// TIA Portal V17 export
// export: Created 2023-12-22T15:05:34.6100322Z, ExportSetting WithDefaults, DisplayName Totally Integrated Automation Portal, DisplayVersion V17, DisplayName TIA Portal Openness, DisplayVersion V17, DisplayName TIA Portal Version Control Interface, DisplayVersion V17, DisplayName STEP 7 Professional, DisplayVersion V17, DisplayName STEP 7 Safety, DisplayVersion V17, DisplayName WinCC Advanced, DisplayVersion V17
DATA_BLOCK "DB_Comm"   // DB99
{ S7_Optimized_Access := 'FALSE' }
VERSION : 0.1
// stored: AutoNumber false, DBAccessibleFromOPCUA true, IsOnlyStoredInLoadMemory false, IsWriteProtectedInAS false
   VAR RETAIN
      Input : Struct
         Line : Array[0..7] of Struct   // Линии
            Start : Bool;   // Дистанционный старт линии
            Mode : Bool;   // 0 - без разбавления, 1 - с разбавлением
            D : Real;   // Доза линии
         END_STRUCT;
         Pump : Array[1..10] of Struct   // Насосы
            Reserv : Bool;   // 0 - насос основной, 1 - насос резервный
            Line_Main : Int;   // Главная линия насоса
            Line_Reserve : Int;   // Резервная линия насоса
         END_STRUCT;
         Input_PolyMix_1 : "PolyMix_Input";
         Input_PolyMix_2 : "PolyMix_Input";
         Flow_LSAU_1 : Real := 1314.753;   // м3/ч
         Flow_LSAU_2 : Real := 0.0;
         Reset_All : Bool := FALSE;
         PolyMix_1_Source_BK1 : Bool := FALSE;   // Жидкий полимикс - качает с бака 1
         PolyMix_1_Source_BK2 : Bool := TRUE;   // Жидкий полимикс - качает с бака 2
         L123_S_P1 : Bool := FALSE;   // Линия 1 - работает жидким полимиксом
         L123_S_P2 : Bool := TRUE;   // Линия 1 - работает с сухим полимиксом
         L456_S_P1 : Bool := TRUE;   // Линия 2 - работает жидким полимиксом
         L456_S_P2 : Bool := FALSE;   // Линия 2 - работает с сухим полимиксом
         Income_Start : Bool := FALSE;   // Запуск приёмки коагулянта
         Income_Line : Bool := FALSE;   // Приёмка с машины
         Income_Pump : Bool := TRUE;   // Приёмка с кубиков
         Income_BK1 : Bool := TRUE;   // Приёмка в бак БК 1
         Income_BK2 : Bool := FALSE;   // Приёмка в бак БК 2
         Recirk_BK1_Use : Bool := TRUE;   // Автоматическая рециркуляция БК 1
         Recirk_BK2_Use : Bool := TRUE;   // Автоматическая рециркуляция БК 2
         Recirk_BK1_Start : Bool := FALSE;   // Запуск рецикруляции БК 1
         Recirk_BK2_Start : Bool := FALSE;   // Запуск рецикруляции БК 2
         "word" : Word := 16#0000;
      END_STRUCT;
      Output : Struct
         Line : Array[0..7] of Struct   // Линии
            Start : Bool;   // 0 - линия выкл, 1 - линия в работе
            Mode : Bool;   // 0 - без разбавления, 1 - с разбавлением
            Local : Bool;   // 0 - местный режим, 1 - дистанционный
            KC : Bool;   // 0 - КС закрыт, 1 - КС открыт
            RT : Bool;   // 0 - нет протока на РТ, 1 - есть проток на РТ
            D : Real;   // Текущая уставка Дозы
         END_STRUCT;
         Pump : Array[1..10] of Struct   // Насосы
            Reserv : Bool;   // 0 - насос основной, 1 - насос резервный
            Status : Int;   // Статус насоса
            SP : Real;   // Скорость работы насоса
            Line_Main : Int;   // Главная линия насоса
            Line_Reserv : Int;   // Резервная линия насоса
         END_STRUCT;
         Output_PolyMix_1 : "PolyMix_Output";
         Output_PolyMix_2 : "PolyMix_Output";
         PolyMix_1_Source_BK1 : Bool := FALSE;   // Жидкий полимикс - качает с бака 1
         PolyMix_1_Source_BK2 : Bool := TRUE;   // Жидкий полимикс - качает с бака 2
         L123_S_P1 : Bool := FALSE;   // Линия 1 - работает жидким полимиксом
         L123_S_P2 : Bool := TRUE;   // Линия 1 - работает с сухим полимиксом
         L456_S_P1 : Bool := TRUE;   // Линия 2 - работает жидким полимиксом
         L456_S_P2 : Bool := FALSE;   // Линия 2 - работает с сухим полимиксом
         Any_Alarm : Bool := FALSE;   // Общая авария
         Income_Start : Bool := FALSE;   // Запуск приёмки коагулянта
         Income_Line : Bool := FALSE;   // Приёмка с машины
         Income_Pump : Bool := TRUE;   // Приёмка с кубиков
         Income_BK1 : Bool := TRUE;   // Приёмка в бак БК 1
         Income_BK2 : Bool := FALSE;   // Приёмка в бак БК 2
         Recirk_BK1_Use : Bool := TRUE;   // Автоматическая рециркуляция БК 1
         Recirk_BK2_Use : Bool := TRUE;   // Автоматическая рециркуляция БК 2
         Recirk_BK1_Start : Bool := FALSE;   // Запуск рецикруляции БК 1
         Recirk_BK2_Start : Bool := FALSE;   // Запуск рецикруляции БК 2
         reserv : Word := 16#0000;
      END_STRUCT;
      Time_DTL : DTL := DTL#2020-10-13-13:05:17.729949026;
   END_VAR
BEGIN
   Input.Line[0..7].Start := FALSE;
   Input.Line[0].Mode := FALSE;
   Input.Line[1..6].Mode := TRUE;
   Input.Line[7].Mode := FALSE;
   Input.Line[0].D := 3.0;
   Input.Line[1..2].D := 1.0E-05;
   Input.Line[3].D := 3.0E-05;
   Input.Line[4].D := 4.0E-05;
   Input.Line[5].D := 5.0E-05;
   Input.Line[6].D := 6.0E-05;
   Input.Line[7].D := 0.1;
   Input.Pump[1..7].Reserv := FALSE;
   Input.Pump[8].Reserv := TRUE;
   Input.Pump[9].Reserv := FALSE;
   Input.Pump[10].Reserv := TRUE;
   Input.Pump[1].Line_Main := 1;
   Input.Pump[2].Line_Main := 2;
   Input.Pump[3].Line_Main := 3;
   Input.Pump[4].Line_Main := 4;
   Input.Pump[5].Line_Main := 5;
   Input.Pump[6].Line_Main := 6;
   Input.Pump[7].Line_Main := 7;
   Input.Pump[8].Line_Main := 0;
   Input.Pump[9].Line_Main := 8;
   Input.Pump[10].Line_Main := 0;
   Input.Pump[1..7].Line_Reserve := 0;
   Input.Pump[8].Line_Reserve := 7;
   Input.Pump[9].Line_Reserve := 0;
   Input.Pump[10].Line_Reserve := 8;
   Input.Input_PolyMix_1.WatchDog := 2985;   // Контроль связи 0...1000 раз в секунду
   Input.Input_PolyMix_1.Clock := FALSE;   // Контроль связи 1 Гц
   Input.Input_PolyMix_1.Start := TRUE;
   Input.Input_PolyMix_1.SP_C := 9.0;
   Input.Input_PolyMix_1.Weight := 0.0;   // Внешние данные о весе
   Input.Input_PolyMix_1.res_1 := 0.0;   // Резерв 1
   Input.Input_PolyMix_1.res_2 := 0.0;   // Резерв 2
   Input.Input_PolyMix_2.WatchDog := 2985;   // Контроль связи 0...1000 раз в секунду
   Input.Input_PolyMix_2.Clock := FALSE;   // Контроль связи 1 Гц
   Input.Input_PolyMix_2.Start := FALSE;
   Input.Input_PolyMix_2.SP_C := 5.0;
   Input.Input_PolyMix_2.Weight := 593.0253;   // Внешние данные о весе
   Input.Input_PolyMix_2.res_1 := 0.0;   // Резерв 1
   Input.Input_PolyMix_2.res_2 := 0.0;   // Резерв 2
   Output.Line[0..7].Start := FALSE;
   Output.Line[0].Mode := FALSE;
   Output.Line[1..6].Mode := TRUE;
   Output.Line[7].Mode := FALSE;
   Output.Line[0].Local := FALSE;
   Output.Line[1..6].Local := TRUE;
   Output.Line[7].Local := FALSE;
   Output.Line[0..7].KC := FALSE;
   Output.Line[0..7].RT := FALSE;
   Output.Line[0].D := 3.0;
   Output.Line[1..2].D := 1.0E-05;
   Output.Line[3].D := 3.0E-05;
   Output.Line[4].D := 4.0E-05;
   Output.Line[5].D := 5.0E-05;
   Output.Line[6].D := 6.0E-05;
   Output.Line[7].D := 0.1;
   Output.Pump[1..7].Reserv := FALSE;
   Output.Pump[8].Reserv := TRUE;
   Output.Pump[9].Reserv := FALSE;
   Output.Pump[10].Reserv := TRUE;
   Output.Pump[1..10].Status := 0;
   Output.Pump[1..10].SP := 0.0;
   Output.Pump[1].Line_Main := 1;
   Output.Pump[2].Line_Main := 2;
   Output.Pump[3].Line_Main := 3;
   Output.Pump[4].Line_Main := 4;
   Output.Pump[5].Line_Main := 5;
   Output.Pump[6].Line_Main := 6;
   Output.Pump[7].Line_Main := 7;
   Output.Pump[8].Line_Main := 0;
   Output.Pump[9].Line_Main := 8;
   Output.Pump[10].Line_Main := 0;
   Output.Pump[1..7].Line_Reserv := 0;
   Output.Pump[8].Line_Reserv := 7;
   Output.Pump[9].Line_Reserv := 0;
   Output.Pump[10].Line_Reserv := 8;
   Output.Output_PolyMix_1.WatchDog := 182;   // Контроль связи 0...1000 раз в секунду
   Output.Output_PolyMix_1.Clock := TRUE;   // Контроль связи 1 Гц
   Output.Output_PolyMix_1.Start := TRUE;
   Output.Output_PolyMix_1.LS_1 := FALSE;
   Output.Output_PolyMix_1.LS_2 := FALSE;
   Output.Output_PolyMix_1.LS_3 := FALSE;
   Output.Output_PolyMix_1.LS_4 := FALSE;
   Output.Output_PolyMix_1.KC_1 := FALSE;
   Output.Output_PolyMix_1.ALLS := FALSE;
   Output.Output_PolyMix_1.Local := FALSE;
   Output.Output_PolyMix_1.LLS := FALSE;
   Output.Output_PolyMix_1.HLS := TRUE;
   Output.Output_PolyMix_1.SP_C := 9.0;
   Output.Output_PolyMix_1.Level := 985.9791;
   Output.Output_PolyMix_1.Flow := 0.0;
   Output.Output_PolyMix_1.Weight := 0.0;   // Внешние данные о весе
   Output.Output_PolyMix_1.Mix_1 := 0;
   Output.Output_PolyMix_1.Mix_2 := 0;
   Output.Output_PolyMix_1.Mix_3 := 0;
   Output.Output_PolyMix_1.SD := 0;
   Output.Output_PolyMix_1.DD := 0;
   Output.Output_PolyMix_1.SH := 0;
   Output.Output_PolyMix_1.PN := 0;
   Output.Output_PolyMix_1.Vibro := 0;
   Output.Output_PolyMix_1.Vent := 0;
   Output.Output_PolyMix_1.Messages.Flow_Dry_Run := FALSE;
   Output.Output_PolyMix_1.Messages.Flow_Low := FALSE;
   Output.Output_PolyMix_1.Messages.LE_NoChange := FALSE;
   Output.Output_PolyMix_1.Messages.LE_Low := FALSE;
   Output.Output_PolyMix_1.Messages.LE_High := FALSE;
   Output.Output_PolyMix_1.Messages.LS_Low := FALSE;
   Output.Output_PolyMix_1.Messages.LS_NoProduct := FALSE;
   Output.Output_PolyMix_1.Messages.LS_Filter := FALSE;
   Output.Output_PolyMix_1.Messages.SD_Low := FALSE;
   Output.Output_PolyMix_1.Messages.Low_Weight := FALSE;
   Output.Output_PolyMix_1.Messages.Link_Error := FALSE;
   Output.Output_PolyMix_1.Messages.Alarm := 16#0000;
   Output.Output_PolyMix_1.Report.C := 0.0;
   Output.Output_PolyMix_1.Report.Water := 0.0;
   Output.Output_PolyMix_1.Report.Reagent := 0.0;
   Output.Output_PolyMix_1.Report.Weight := 0.0;
   Output.Output_PolyMix_1.Report.Dos := 0.0;
   Output.Output_PolyMix_1.Report.Res := 0.0;
   Output.Output_PolyMix_1.Report.WeekDay := 2;
   Output.Output_PolyMix_1.Report.Day := 12;
   Output.Output_PolyMix_1.Report.Month := 10;
   Output.Output_PolyMix_1.LE_Alarm := 16#0000;
   Output.Output_PolyMix_2.WatchDog := 182;   // Контроль связи 0...1000 раз в секунду
   Output.Output_PolyMix_2.Clock := TRUE;   // Контроль связи 1 Гц
   Output.Output_PolyMix_2.Start := FALSE;
   Output.Output_PolyMix_2.LS_1 := FALSE;
   Output.Output_PolyMix_2.LS_2 := TRUE;
   Output.Output_PolyMix_2.LS_3 := FALSE;
   Output.Output_PolyMix_2.LS_4 := FALSE;
   Output.Output_PolyMix_2.KC_1 := FALSE;
   Output.Output_PolyMix_2.ALLS := FALSE;
   Output.Output_PolyMix_2.Local := FALSE;
   Output.Output_PolyMix_2.LLS := FALSE;
   Output.Output_PolyMix_2.HLS := TRUE;
   Output.Output_PolyMix_2.SP_C := 5.0;
   Output.Output_PolyMix_2.Level := 916.5723;
   Output.Output_PolyMix_2.Flow := 0.0;
   Output.Output_PolyMix_2.Weight := 593.0253;   // Внешние данные о весе
   Output.Output_PolyMix_2.Mix_1 := 1;
   Output.Output_PolyMix_2.Mix_2 := 1;
   Output.Output_PolyMix_2.Mix_3 := 1;
   Output.Output_PolyMix_2.SD := 0;
   Output.Output_PolyMix_2.DD := 0;
   Output.Output_PolyMix_2.SH := 0;
   Output.Output_PolyMix_2.PN := 0;
   Output.Output_PolyMix_2.Vibro := 0;
   Output.Output_PolyMix_2.Vent := 0;
   Output.Output_PolyMix_2.Messages.Flow_Dry_Run := FALSE;
   Output.Output_PolyMix_2.Messages.Flow_Low := FALSE;
   Output.Output_PolyMix_2.Messages.LE_NoChange := FALSE;
   Output.Output_PolyMix_2.Messages.LE_Low := FALSE;
   Output.Output_PolyMix_2.Messages.LE_High := FALSE;
   Output.Output_PolyMix_2.Messages.LS_Low := FALSE;
   Output.Output_PolyMix_2.Messages.LS_NoProduct := FALSE;
   Output.Output_PolyMix_2.Messages.LS_Filter := FALSE;
   Output.Output_PolyMix_2.Messages.SD_Low := FALSE;
   Output.Output_PolyMix_2.Messages.Low_Weight := FALSE;
   Output.Output_PolyMix_2.Messages.Link_Error := FALSE;
   Output.Output_PolyMix_2.Messages.Alarm := 16#0000;
   Output.Output_PolyMix_2.Report.C := 5.0;
   Output.Output_PolyMix_2.Report.Water := 1926.197;
   Output.Output_PolyMix_2.Report.Reagent := 321.0332;
   Output.Output_PolyMix_2.Report.Weight := 0.0;
   Output.Output_PolyMix_2.Report.Dos := 10.0;
   Output.Output_PolyMix_2.Report.Res := 0.0;
   Output.Output_PolyMix_2.Report.WeekDay := 2;
   Output.Output_PolyMix_2.Report.Day := 12;
   Output.Output_PolyMix_2.Report.Month := 10;
   Output.Output_PolyMix_2.LE_Alarm := 16#0000;
END_DATA_BLOCK
